// TIA Portal project "babu_PumpValveMixer" (V15)

(* hardware
DEVICE "S7-1200 station_1"  S7-1200 Station
   slot 0: "Rack_0"  S7-1200 Rack  Rack  V1.0
   slot 1: "PLC_1"  CPU 1212C DC/DC/DC  6ES7 212-1AE40-0XB0  V4.2
DEVICE "S7-1200 station_2"  S7-1200 Station
   slot 0: "Rack_0"  S7-1200 Rack  Rack  V1.0
   slot 1: "PLC_2"  CPU 1211C DC/DC/DC  6ES7 211-1AE40-0XB0  V4.2
*)

// ===== PLC "PLC_1"  CPU 1212C DC/DC/DC =====

VAR_GLOBAL   // PLC tag table "Default tag table"
   "Tank" AT %Q0.0 : Bool;
END_VAR

VAR_GLOBAL   // PLC tag table "Tag table_1"
   "PUSH BUTTON" AT %M0.0 : Bool;
   "PUSH BUTTON - MEMORY" AT %M0.1 : Bool;
   "PUMP 1" AT %Q0.2 : Bool;
   "VALVE 1" AT %Q0.3 : Bool;
   "VALVE 2" AT %Q0.4 : Bool;
   "MIXER" AT %Q0.5 : Bool;
   "PUMP 2" AT %Q0.6 : Bool;
   "PUMP 1 MEMORY" AT %M0.7 : Bool;
   "PUMP 2 MEMORY" AT %M1.0 : Bool;
END_VAR

// folder: System blocks/Program resources

DATA_BLOCK "IEC_Timer_0_DB"   // DB1
{ S7_Optimized_Access := 'TRUE' }
AUTHOR : Simatic
FAMILY : IEC
NAME : IEC_TMR
VERSION : 1.0
// stored: InstanceOfName IEC_TIMER
"IEC_TIMER"
BEGIN
END_DATA_BLOCK

DATA_BLOCK "IEC_Timer_0_DB_1"   // DB2
{ S7_Optimized_Access := 'TRUE' }
AUTHOR : Simatic
FAMILY : IEC
NAME : IEC_TMR
VERSION : 1.0
// stored: InstanceOfName IEC_TIMER
"IEC_TIMER"
BEGIN
END_DATA_BLOCK

DATA_BLOCK "IEC_Timer_0_DB_2"   // DB3
{ S7_Optimized_Access := 'TRUE' }
AUTHOR : Simatic
FAMILY : IEC
NAME : IEC_TMR
VERSION : 1.0
// stored: InstanceOfName IEC_TIMER
"IEC_TIMER"
BEGIN
END_DATA_BLOCK

DATA_BLOCK "IEC_Timer_0_DB_3"   // DB4
{ S7_Optimized_Access := 'TRUE' }
AUTHOR : Simatic
FAMILY : IEC
NAME : IEC_TMR
VERSION : 1.0
// stored: InstanceOfName IEC_TIMER
"IEC_TIMER"
BEGIN
END_DATA_BLOCK

DATA_BLOCK "IEC_Timer_0_DB_4"   // DB5
{ S7_Optimized_Access := 'TRUE' }
AUTHOR : Simatic
FAMILY : IEC
NAME : IEC_TMR
VERSION : 1.0
// stored: InstanceOfName IEC_TIMER
"IEC_TIMER"
BEGIN
END_DATA_BLOCK

// folder: (top level)

ORGANIZATION_BLOCK "Main"   // OB1, LAD, ProgramCycle
TITLE = "Main Program Sweep (Cycle)"
{ S7_Optimized_Access := 'TRUE' }
VERSION : 0.1
   VAR_INPUT
      Initial_Call : Bool;   // Initial call of this OB
      Remanence : Bool;   // =True, if remanent data are available
   END_VAR
BEGIN

REGION Network 1
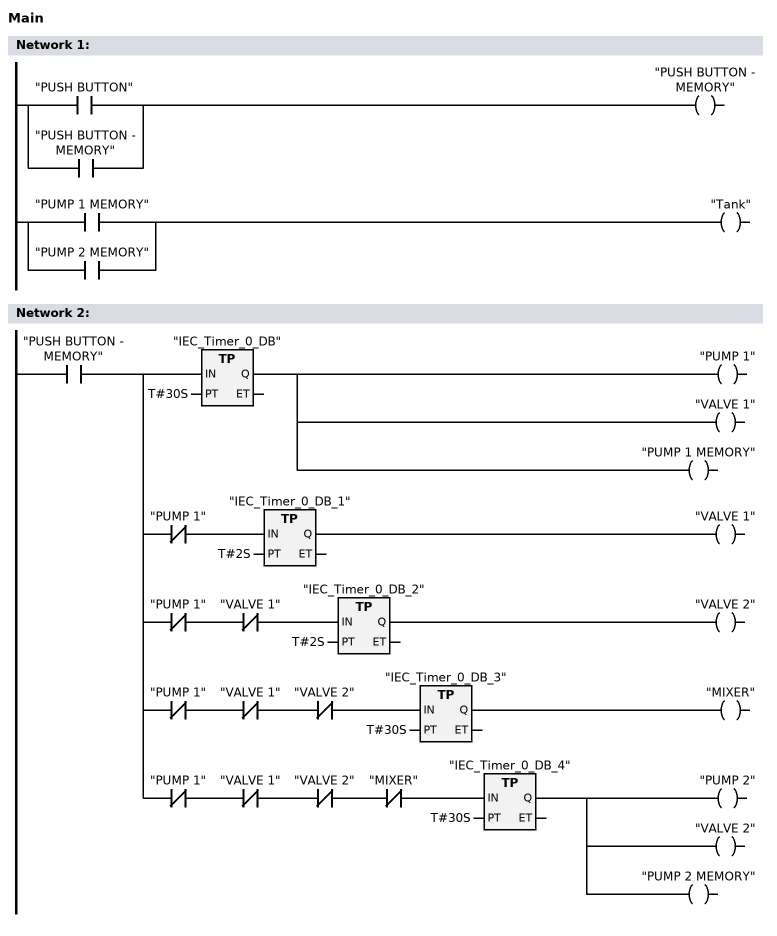
   RUNG wire#powerrail
      Contact( "PUSH BUTTON" )
      wire#w1
      Coil( "PUSH BUTTON - MEMORY" )
   END_RUNG
   RUNG wire#powerrail
      Contact( "PUSH BUTTON - MEMORY" )
   END_RUNG wire#w1
   RUNG wire#powerrail
      Contact( "PUMP 1 MEMORY" )
      wire#w2
      Coil( "Tank" )
   END_RUNG
   RUNG wire#powerrail
      Contact( "PUMP 2 MEMORY" )
   END_RUNG wire#w2
   // the same network as SCL:
   "PUSH BUTTON - MEMORY" := "PUSH BUTTON" OR "PUSH BUTTON - MEMORY";
   "Tank" := "PUMP 1 MEMORY" OR "PUMP 2 MEMORY";
END_REGION

REGION Network 2
   "IEC_Timer_0_DB".TP(IN := "PUSH BUTTON - MEMORY", PT := T#30S);
   "PUMP 1" := "IEC_Timer_0_DB".Q;
   "VALVE 1" := "IEC_Timer_0_DB".Q;
   "PUMP 1 MEMORY" := "IEC_Timer_0_DB".Q;
   "IEC_Timer_0_DB_1".TP(IN := "PUSH BUTTON - MEMORY" AND NOT "PUMP 1", PT := T#2S);
   "VALVE 1" := "IEC_Timer_0_DB_1".Q;
   "IEC_Timer_0_DB_2".TP(IN := "PUSH BUTTON - MEMORY" AND NOT "PUMP 1" AND NOT "VALVE 1", PT := T#2S);
   "VALVE 2" := "IEC_Timer_0_DB_2".Q;
   "IEC_Timer_0_DB_3".TP(IN := "PUSH BUTTON - MEMORY" AND NOT "PUMP 1" AND NOT "VALVE 1" AND NOT "VALVE 2",
                         PT := T#30S);
   "MIXER" := "IEC_Timer_0_DB_3".Q;
   "IEC_Timer_0_DB_4".TP(IN := "PUSH BUTTON - MEMORY" AND NOT "PUMP 1" AND NOT "VALVE 1" AND NOT "VALVE 2" AND NOT "MIXER",
                         PT := T#30S);
   "PUMP 2" := "IEC_Timer_0_DB_4".Q;
   "VALVE 2" := "IEC_Timer_0_DB_4".Q;
   "PUMP 2 MEMORY" := "IEC_Timer_0_DB_4".Q;
END_REGION
END_ORGANIZATION_BLOCK

// ===== PLC "PLC_2"  CPU 1211C DC/DC/DC =====

ORGANIZATION_BLOCK "Main"   // OB1, LAD, ProgramCycle
TITLE = "Main Program Sweep (Cycle)"
{ S7_Optimized_Access := 'TRUE' }
VERSION : 0.1
   VAR_INPUT
      Initial_Call : Bool;   // Initial call of this OB
      Remanence : Bool;   // =True, if remanent data are available
   END_VAR
BEGIN
END_ORGANIZATION_BLOCK